// TIA Portal V17 export
// export: Created 2024-08-26T21:10:51.0363505Z, ExportSetting WithDefaults, DisplayName Totally Integrated Automation Portal, DisplayVersion V17 Update 7, DisplayName TIA Portal Openness, DisplayVersion V17 Update 7, DisplayName TIA Portal Version Control Interface, DisplayVersion V17, DisplayName SINAMICS Startdrive Advanced, DisplayVersion V17 SP2, DisplayName SINAMICS Startdrive G110M, G120, G120C, G120D, G120P, G115D, DisplayVersion V17 SP2, DisplayName SINAMICS Startdrive G130, G150, S120, S150, SINAMICS MV, S210, DisplayVersion V17 SP2, DisplayName STEP 7 Professional, DisplayVersion V17 Update 7, DisplayName STEP 7 Safety, DisplayVersion V17 Update 6, DisplayName WinCC Advanced / Unified PC, DisplayVersion V17 Update 7
FUNCTION_BLOCK "Time System"   // FB2420, LAD
{ S7_Optimized_Access := 'TRUE' }
VERSION : 0.1
// stored: AutoNumber false, IsIECCheckEnabled false, IsRetainMemResEnabled false, MemoryReserve 100, SetENOAutomatically false, UDAEnableTagReadback false
   VAR_INPUT
      bPartOkNok : Bool;
      bRunningcycle : Bool;
      bPreCount : Bool;
   END_VAR
   VAR_OUTPUT
      bShift1 : Bool;
      bShift2 : Bool;
      bShift3 : Bool;
      nCycle_Time_Shift : Real;
      nCycleTimeAvg_Shift1 : Real;
      nCycleTimeAvg_Shift2 : Real;
      nCycleTimeAvg_Shift3 : Real;
   END_VAR
   VAR
      Ret_Val_WR { ExternalAccessible := 'False'; ExternalVisible := 'False'; ExternalWritable := 'False'} : USInt;
      Ret_Val_RD { ExternalAccessible := 'False'; ExternalVisible := 'False'; ExternalWritable := 'False'} : USInt;
      DTL_Set_Time : DTL;
      DTL_Read_Time : DTL;
      TOD_Read : Time_Of_Day;
      Date_Read : Date;
      bAceptButtonHmiP : Bool;
      bAcept_buttonHMI : Bool;
      nSet_minute : Int;
      nSet_Hour : Int;
      nSet_Day : Int;
      nSet_Month : Int;
      nSet_Year : Int;
      nCycleTimeArray : Array[0..5] of Real;
      tCycleTime { S7_SetPoint := 'True'} : IEC_TIMER;
      nCycleTimeET : UDInt;
      tCycleTimeTotal : UDInt;
      bPartOkNokP : Bool;
      bPartOkNokCmd : Bool;
      nPartAvgCounter : Int;
      bCycle_StartedP : Bool;
      bSH1 : Bool;
      bSH2 : Bool;
      bSH3 : Bool;
      nCycle_Time : Real;
      nCycleTimeAvg : Real;
      Read_Local_Time : DTL;
      Read_System_Time : DTL;
      Time_HMI_Set : DTL;
      RetVal1 : Word;
      Retval2 : Word;
      Retval3 : Word;
      n : Int;
      timesCounter { S7_SetPoint := 'True'} : IEC_COUNTER;
   END_VAR
   VAR RETAIN
      tCycle_Running : Real;
   END_VAR
   VAR
      nCycleAvg : DInt;
      nCycleTime_Total : Time_Of_Day;
      ntimeRun_conv : UDInt;
   END_VAR
   // nCycleTimeArray[3..5] := 0.0;
   VAR_TEMP   // added for the SCL form of the ladder/FBD networks
      _w1 : Bool;
   END_VAR
BEGIN

REGION Network 1: SET HOUR
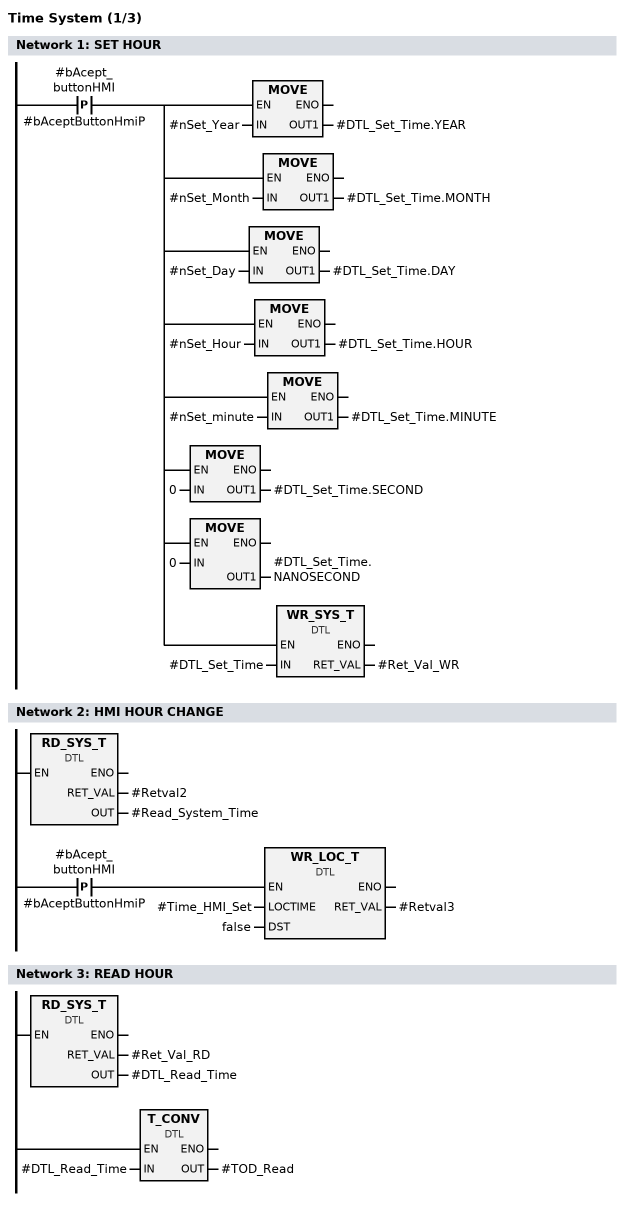
   RUNG wire#powerrail
      P_Contact(operand := #bAcept_buttonHMI, bit := #bAceptButtonHmiP)
      wire#w1
      Move(in := #nSet_Year, out1 => #DTL_Set_Time.YEAR)
   END_RUNG
   RUNG wire#w1
      Move(in := #nSet_Month, out1 => #DTL_Set_Time.MONTH)
   END_RUNG
   RUNG wire#w1
      Move(in := #nSet_Day, out1 => #DTL_Set_Time.DAY)
   END_RUNG
   RUNG wire#w1
      Move(in := #nSet_Hour, out1 => #DTL_Set_Time.HOUR)
   END_RUNG
   RUNG wire#w1
      Move(in := #nSet_minute, out1 => #DTL_Set_Time.MINUTE)
   END_RUNG
   RUNG wire#w1
      Move(in := 0, out1 => #DTL_Set_Time.SECOND)
   END_RUNG
   RUNG wire#w1
      Move(in := 0, out1 => #DTL_Set_Time.NANOSECOND)
   END_RUNG
   RUNG wire#w1
      { S7_Templates := "date_type := DTL" } WR_SYS_T(IN := #DTL_Set_Time, RET_VAL => #Ret_Val_WR)
   END_RUNG
   // the same network as SCL:
   #_w1 := #bAcept_buttonHMI AND NOT #bAceptButtonHmiP;   // rising edge of #bAcept_buttonHMI
   #bAceptButtonHmiP := #bAcept_buttonHMI;
   IF #_w1 THEN
       #DTL_Set_Time.YEAR := #nSet_Year;
       #DTL_Set_Time.MONTH := #nSet_Month;
       #DTL_Set_Time.DAY := #nSet_Day;
       #DTL_Set_Time.HOUR := #nSet_Hour;
       #DTL_Set_Time.MINUTE := #nSet_minute;
       #DTL_Set_Time.SECOND := 0;
       #DTL_Set_Time.NANOSECOND := 0;
       #Ret_Val_WR := WR_SYS_T(IN := #DTL_Set_Time);
   END_IF;
END_REGION

REGION Network 2: HMI HOUR CHANGE
   RUNG wire#powerrail
      { S7_Templates := "date_type := DTL" } RD_SYS_T(RET_VAL => #Retval2, OUT => #Read_System_Time)
   END_RUNG
   RUNG wire#powerrail
      P_Contact(operand := #bAcept_buttonHMI, bit := #bAceptButtonHmiP)
      { S7_Templates := "loctime_type := DTL" } WR_LOC_T(LOCTIME := #Time_HMI_Set, DST := false, Ret_Val => #Retval3)
   END_RUNG
   // the same network as SCL:
   #Retval2 := RD_SYS_T(OUT => #Read_System_Time);
   #_w1 := #bAcept_buttonHMI AND NOT #bAceptButtonHmiP;   // rising edge of #bAcept_buttonHMI
   #bAceptButtonHmiP := #bAcept_buttonHMI;
   IF #_w1 THEN #Retval3 := WR_LOC_T(LOCTIME := #Time_HMI_Set, DST := false); END_IF;
END_REGION

REGION Network 3: READ HOUR
   RUNG wire#powerrail
      { S7_Templates := "date_type := DTL" } RD_SYS_T(RET_VAL => #Ret_Val_RD, OUT => #DTL_Read_Time)
   END_RUNG
   RUNG wire#powerrail
      { S7_Templates := "[src_type := DTL, dest_type := Time_Of_Day]" } T_CONV(IN := #DTL_Read_Time, OUT => #TOD_Read)
   END_RUNG
   // the same network as SCL:
   #Ret_Val_RD := RD_SYS_T(OUT => #DTL_Read_Time);
   T_CONV(IN := #DTL_Read_Time, OUT => #TOD_Read);
END_REGION

REGION Network 4: WORK SHIFTS
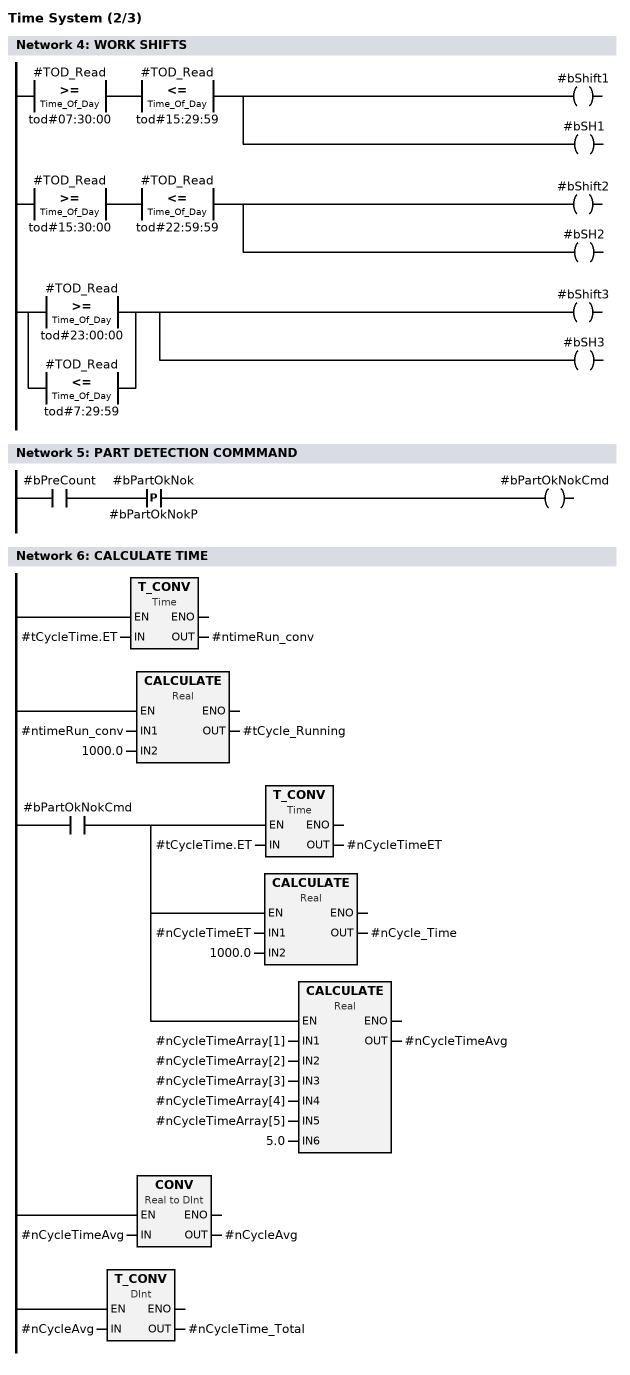
   RUNG wire#powerrail
      { S7_Templates := "SrcType := Time_Of_Day" } GE_Contact(in1 := #TOD_Read, in2 := tod#07:30:00)
      { S7_Templates := "SrcType := Time_Of_Day" } LE_Contact(in1 := #TOD_Read, in2 := tod#15:29:59)
      wire#w1
      Coil( #bShift1 )
   END_RUNG
   RUNG wire#w1
      Coil( #bSH1 )
   END_RUNG
   RUNG wire#powerrail
      { S7_Templates := "SrcType := Time_Of_Day" } GE_Contact(in1 := #TOD_Read, in2 := tod#15:30:00)
      { S7_Templates := "SrcType := Time_Of_Day" } LE_Contact(in1 := #TOD_Read, in2 := tod#22:59:59)
      wire#w2
      Coil( #bShift2 )
   END_RUNG
   RUNG wire#w2
      Coil( #bSH2 )
   END_RUNG
   RUNG wire#powerrail
      { S7_Templates := "SrcType := Time_Of_Day" } GE_Contact(in1 := #TOD_Read, in2 := tod#23:00:00)
      wire#w3
      Coil( #bShift3 )
   END_RUNG
   RUNG wire#powerrail
      { S7_Templates := "SrcType := Time_Of_Day" } LE_Contact(in1 := #TOD_Read, in2 := tod#7:29:59)
   END_RUNG wire#w3
   RUNG wire#w3
      Coil( #bSH3 )
   END_RUNG
   // the same network as SCL:
   #bShift1 := (#TOD_Read >= tod#07:30:00) AND (#TOD_Read <= tod#15:29:59);
   #bSH1 := #bShift1;
   #bShift2 := (#TOD_Read >= tod#15:30:00) AND (#TOD_Read <= tod#22:59:59);
   #bSH2 := #bShift2;
   #bShift3 := (#TOD_Read >= tod#23:00:00) OR (#TOD_Read <= tod#7:29:59);
   #bSH3 := #bShift3;
END_REGION

REGION Network 5: PART DETECTION COMMMAND
   RUNG wire#powerrail
      Contact( #bPreCount )
      P_Contact(operand := #bPartOkNok, bit := #bPartOkNokP)
      Coil( #bPartOkNokCmd )
   END_RUNG
   // the same network as SCL:
   #_w1 := #bPreCount AND #bPartOkNok AND NOT #bPartOkNokP;   // rising edge of #bPartOkNok
   #bPartOkNokP := #bPartOkNok;
   #bPartOkNokCmd := #_w1;
END_REGION

REGION Network 6: CALCULATE TIME
   RUNG wire#powerrail
      { S7_Templates := "[src_type := Time, dest_type := UDInt]" } T_CONV(IN := #tCycleTime.ET, OUT => #ntimeRun_conv)
   END_RUNG
   RUNG wire#powerrail
      { S7_Templates := "SrcType := Real"; S7_Expression := "in1/in2" } Calculate(in1 := #ntimeRun_conv, in2 := 1000.0, out => #tCycle_Running)
   END_RUNG
   RUNG wire#powerrail
      Contact( #bPartOkNokCmd )
      wire#w1
      { S7_Templates := "[src_type := Time, dest_type := UDInt]" } T_CONV(IN := #tCycleTime.ET, OUT => #nCycleTimeET)
   END_RUNG
   RUNG wire#w1
      { S7_Templates := "SrcType := Real"; S7_Expression := "in1/in2" } Calculate(in1 := #nCycleTimeET, in2 := 1000.0, out => #nCycle_Time)
   END_RUNG
   RUNG wire#w1
      { S7_Templates := "SrcType := Real"; S7_Expression := "(in1+in2+in3+in4+in5)/in6" } Calculate(in1 := #nCycleTimeArray[1], in2 := #nCycleTimeArray[2], in3 := #nCycleTimeArray[3], in4 := #nCycleTimeArray[4], in5 := #nCycleTimeArray[5], in6 := 5.0, out => #nCycleTimeAvg)
   END_RUNG
   RUNG wire#powerrail
      { S7_Templates := "[SrcType := Real, DestType := DInt]" } Convert(in := #nCycleTimeAvg, out => #nCycleAvg)
   END_RUNG
   RUNG wire#powerrail
      { S7_Templates := "[src_type := DInt, dest_type := Time_Of_Day]" } T_CONV(IN := #nCycleAvg, OUT => #nCycleTime_Total)
   END_RUNG
   // the same network as SCL:
   T_CONV(IN := #tCycleTime.ET, OUT => #ntimeRun_conv);
   #tCycle_Running := #ntimeRun_conv/1000.0;
   IF #bPartOkNokCmd THEN
       T_CONV(IN := #tCycleTime.ET, OUT => #nCycleTimeET);
       #nCycle_Time := #nCycleTimeET/1000.0;
       #nCycleTimeAvg := (#nCycleTimeArray[1]+#nCycleTimeArray[2]+#nCycleTimeArray[3]+#nCycleTimeArray[4]+#nCycleTimeArray[5])/5.0;
   END_IF;
   #nCycleAvg := REAL_TO_DINT(#nCycleTimeAvg);
   T_CONV(IN := #nCycleAvg, OUT => #nCycleTime_Total);
END_REGION

REGION Network 7: CICLE TIME ARRANGEMENT
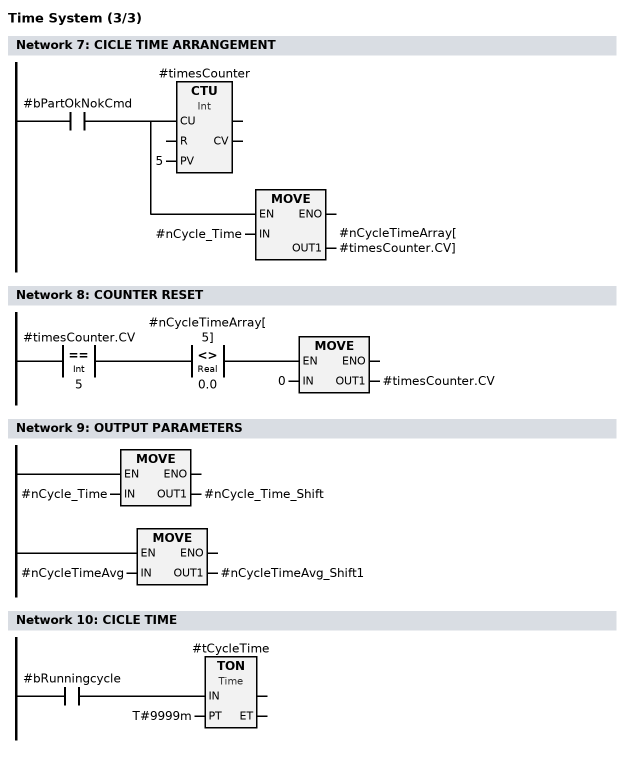
   RUNG wire#powerrail
      Contact( #bPartOkNokCmd )
      wire#w1
      { S7_Templates := "value_type := Int" } #timesCounter.CTU(r :=, pv := 5, cv =>)
   END_RUNG
   RUNG wire#w1
      Move(in := #nCycle_Time, out1 => #nCycleTimeArray[#timesCounter.CV])
   END_RUNG
   // the same network as SCL:
   #timesCounter.CTU(CU := #bPartOkNokCmd, PV := 5);
   IF #bPartOkNokCmd THEN #nCycleTimeArray[#timesCounter.CV] := #nCycle_Time; END_IF;
END_REGION

REGION Network 8: COUNTER RESET
   RUNG wire#powerrail
      { S7_Templates := "SrcType := Int" } EQ_Contact(in1 := #timesCounter.CV, in2 := 5)
      { S7_Templates := "SrcType := Real" } NE_Contact(in1 := #nCycleTimeArray[5], in2 := 0.0)
      Move(in := 0, out1 => #timesCounter.CV)
   END_RUNG
   // the same network as SCL:
   IF (#timesCounter.CV = 5) AND (#nCycleTimeArray[5] <> 0.0) THEN #timesCounter.CV := 0; END_IF;
END_REGION

REGION Network 9: OUTPUT PARAMETERS
   RUNG wire#powerrail
      Move(in := #nCycle_Time, out1 => #nCycle_Time_Shift)
   END_RUNG
   RUNG wire#powerrail
      Move(in := #nCycleTimeAvg, out1 => #nCycleTimeAvg_Shift1)
   END_RUNG
   // the same network as SCL:
   #nCycle_Time_Shift := #nCycle_Time;
   #nCycleTimeAvg_Shift1 := #nCycleTimeAvg;
END_REGION

REGION Network 10: CICLE TIME
   RUNG wire#powerrail
      Contact( #bRunningcycle )
      { S7_Templates := "time_type := Time" } #tCycleTime.TON(pt := T#9999m, et =>)
   END_RUNG
   // the same network as SCL:
   #tCycleTime.TON(IN := #bRunningcycle, PT := T#9999m);
END_REGION
END_FUNCTION_BLOCK
